Yaskawa INFORM job: ARGAZ7.JBI

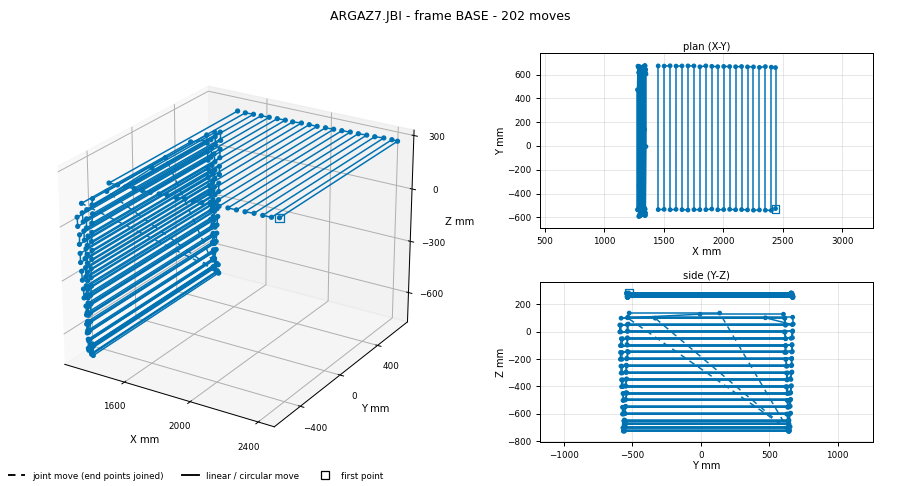
[picture p0: tool path of ARGAZ7.JBI in frame BASE, 202 of 208 moves have a stored position in this frame; points joined in program order, loops and branches not executed]
/JOB
//NAME ARGAZ7
//POS
///NPOS 202,0,202,0,0,0
///TOOL 0
///POSTYPE BASE
///RECTAN
///RCONF 1,0,0,0,0,0,0,0,0,0,0,0,0,0,0,0,0,0,0,0,0,0,0,0
C00000=2438.206271,-525.697965,282.313487,175.000000,5.000000,5.000000
C00001=2438.206271,658.166328,282.313487,175.000000,5.000000,5.000000
C00002=2403.104531,661.654143,282.437479,175.000000,5.000000,5.000000
C00003=2403.104531,-541.268813,282.437479,175.000000,5.000000,5.000000
C00004=2353.104531,-539.692706,280.280820,175.000000,5.000000,5.000000
C00005=2353.104531,666.367518,280.280820,175.000000,5.000000,5.000000
C00006=2303.104531,659.842979,278.975224,175.000000,5.000000,5.000000
C00007=2303.104531,-537.369308,278.975224,175.000000,5.000000,5.000000
C00008=2253.104531,-539.325854,276.432507,175.000000,5.000000,5.000000
C00009=2253.104531,663.877677,276.432507,175.000000,5.000000,5.000000
C00010=2203.104531,664.095750,273.988823,175.000000,5.000000,5.000000
C00011=2203.104531,-536.808159,273.988823,175.000000,5.000000,5.000000
C00012=2153.104531,-534.305410,272.087713,175.000000,5.000000,5.000000
C00013=2153.104531,667.128397,272.087713,175.000000,5.000000,5.000000
C00014=2103.104531,665.272395,270.104448,175.000000,5.000000,5.000000
C00015=2103.104531,-535.482055,270.104448,175.000000,5.000000,5.000000
C00016=2053.104531,-532.207558,267.676633,175.000000,5.000000,5.000000
C00017=2053.104531,666.894698,267.676633,175.000000,5.000000,5.000000
C00018=2003.104531,667.621610,265.646124,175.000000,5.000000,5.000000
C00019=2003.104531,-533.994265,265.646124,175.000000,5.000000,5.000000
C00020=1953.104531,-535.817658,264.262638,175.000000,5.000000,5.000000
C00021=1953.104531,665.764249,264.262638,175.000000,5.000000,5.000000
C00022=1903.104531,668.606677,262.597691,175.000000,5.000000,5.000000
C00023=1903.104531,-529.609020,262.597691,175.000000,5.000000,5.000000
C00024=1853.104531,-535.014658,260.699220,175.000000,5.000000,5.000000
C00025=1853.104531,672.443681,260.699220,175.000000,5.000000,5.000000
C00026=1803.104531,665.010164,259.433234,175.000000,5.000000,5.000000
C00027=1803.104531,-534.903244,259.433234,175.000000,5.000000,5.000000
C00028=1753.104531,-534.503782,257.000030,175.000000,5.000000,5.000000
C00029=1753.104531,672.230363,257.000030,175.000000,5.000000,5.000000
C00030=1703.104531,672.470856,255.326633,175.000000,5.000000,5.000000
C00031=1703.104531,-538.010620,255.326633,175.000000,5.000000,5.000000
C00032=1653.104531,-534.934494,253.475396,175.000000,5.000000,5.000000
C00033=1653.104531,671.829543,253.475396,175.000000,5.000000,5.000000
C00034=1603.104531,670.609419,252.672149,175.000000,5.000000,5.000000
C00035=1603.104531,-532.412044,252.672149,175.000000,5.000000,5.000000
C00036=1553.104531,-535.348902,250.461758,175.000000,5.000000,5.000000
C00037=1553.104531,673.341791,250.461758,175.000000,5.000000,5.000000
C00038=1503.104531,670.724910,249.387708,175.000000,5.000000,5.000000
C00039=1503.104531,-532.359734,249.387708,175.000000,5.000000,5.000000
C00040=1453.054088,-534.367911,249.591599,175.000000,5.000000,5.000000
C00041=1453.054088,672.087699,249.591599,175.000000,5.000000,5.000000
C00042=1350.381240,603.865126,127.297248,175.000000,-89.999999,5.000000
C00043=1350.381240,-4.872901,127.297248,175.000000,-89.999999,5.000000
C00044=1345.317967,-581.433967,98.136038,175.000000,-89.999999,5.000000
C00045=1345.317967,614.304117,98.136038,175.000000,-89.999999,5.000000
C00046=1343.165957,618.982165,48.136038,175.000000,-89.999999,5.000000
C00047=1343.165957,-582.765505,48.136038,175.000000,-89.999999,5.000000
C00048=1341.300612,-583.336165,-1.863962,175.000000,-89.999999,5.000000
C00049=1341.300612,609.146443,-1.863962,175.000000,-89.999999,5.000000
C00050=1339.709084,619.520215,-51.863962,175.000000,-89.999999,5.000000
C00051=1339.709084,-570.470513,-51.863962,175.000000,-89.999999,5.000000
C00052=1337.699081,-576.338794,-101.863962,175.000000,-89.999999,5.000000
C00053=1337.699081,621.164257,-101.863962,175.000000,-89.999999,5.000000
C00054=1336.029732,622.134378,-151.863962,175.000000,-89.999999,5.000000
C00055=1336.029732,-575.046658,-151.863962,175.000000,-89.999999,5.000000
C00056=1334.409462,-575.048017,-201.863962,175.000000,-89.999999,5.000000
C00057=1334.409462,620.847677,-201.863962,175.000000,-89.999999,5.000000
C00058=1332.613520,629.372241,-251.863962,175.000000,-89.999999,5.000000
C00059=1332.613520,-574.966494,-251.863962,175.000000,-89.999999,5.000000
C00060=1330.809111,-573.285766,-301.863962,175.000000,-89.999999,5.000000
C00061=1330.809111,633.836971,-301.863962,175.000000,-89.999999,5.000000
C00062=1328.972483,628.403479,-351.863962,175.000000,-89.999999,5.000000
C00063=1328.972483,-568.874026,-351.863962,175.000000,-89.999999,5.000000
C00064=1327.018956,-568.863156,-401.863962,175.000000,-89.999999,5.000000
C00065=1327.018956,630.494538,-401.863962,175.000000,-89.999999,5.000000
C00066=1325.088817,639.463401,-451.863962,175.000000,-89.999999,5.000000
C00067=1325.088817,-566.032958,-451.863962,175.000000,-89.999999,5.000000
C00068=1323.161118,-565.087294,-501.863962,175.000000,-89.999999,5.000000
C00069=1323.161118,635.588352,-501.863962,175.000000,-89.999999,5.000000
C00070=1321.094332,638.798990,-551.863962,175.000000,-89.999999,5.000000
C00071=1321.094332,-562.729927,-551.863962,175.000000,-89.999999,5.000000
C00072=1319.309806,-563.197324,-601.863962,175.000000,-89.999999,5.000000
C00073=1319.309806,636.908341,-601.863962,175.000000,-89.999999,5.000000
C00074=1317.380318,638.679424,-651.863962,175.000000,-89.999999,5.000000
C00075=1317.380318,-558.654468,-651.863962,175.000000,-89.999999,5.000000
C00076=1315.669137,-556.653763,-701.863962,175.000000,-89.999999,5.000000
C00077=1315.669137,640.156344,-701.863962,175.000000,-89.999999,5.000000
C00078=1334.065119,643.160458,-676.863962,180.000000,-60.000000,0.000000
C00079=1334.065119,-555.617066,-676.863962,180.000000,-60.000000,0.000000
C00080=1332.634857,-557.949975,-726.863962,180.000000,-60.000000,0.000000
C00081=1332.634857,645.315377,-726.863962,180.000000,-60.000000,0.000000
C00082=1332.634857,645.315377,-726.863962,180.000000,-60.000000,0.000000
C00083=1339.573268,138.476508,135.649167,175.000000,-89.999999,5.000000
C00084=1339.573268,-522.212780,135.649167,175.000000,-89.999999,5.000000
C00085=1342.134154,-531.684245,105.452509,175.000000,-89.999999,5.000000
C00086=1342.134154,671.005872,105.452509,175.000000,-89.999999,5.000000
C00087=1341.644946,675.400567,55.452509,175.000000,-89.999999,5.000000
C00088=1341.644946,-528.175842,55.452509,175.000000,-89.999999,5.000000
C00089=1340.416342,-534.347202,5.452509,175.000000,-89.999999,5.000000
C00090=1340.416342,670.993620,5.452509,175.000000,-89.999999,5.000000
C00091=1339.530292,669.673033,-44.547491,175.000000,-89.999999,5.000000
C00092=1339.530292,-535.215794,-44.547491,175.000000,-89.999999,5.000000
C00093=1338.211943,-538.702415,-94.547491,175.000000,-89.999999,5.000000
C00094=1338.211943,666.424662,-94.547491,175.000000,-89.999999,5.000000
C00095=1337.029328,668.773128,-144.547491,175.000000,-89.999999,5.000000
C00096=1337.029328,-535.105518,-144.547491,175.000000,-89.999999,5.000000
C00097=1335.742282,-538.419237,-194.547491,175.000000,-89.999999,5.000000
C00098=1335.742282,664.151075,-194.547491,175.000000,-89.999999,5.000000
C00099=1334.317615,664.923005,-244.547491,175.000000,-89.999999,5.000000
C00100=1334.317615,-543.588585,-244.547491,175.000000,-89.999999,5.000000
C00101=1332.622991,-545.482334,-294.547491,175.000000,-89.999999,5.000000
C00102=1332.622991,665.844693,-294.547491,175.000000,-89.999999,5.000000
C00103=1330.725701,651.986702,-344.547491,175.000000,-89.999999,5.000000
C00104=1330.725701,-540.830329,-344.547491,175.000000,-89.999999,5.000000
C00105=1328.930857,-548.962147,-394.547491,175.000000,-89.999999,5.000000
C00106=1328.930857,662.201508,-394.547491,175.000000,-89.999999,5.000000
C00107=1326.931876,657.022630,-444.547491,175.000000,-89.999999,5.000000
C00108=1326.931876,-544.291083,-444.547491,175.000000,-89.999999,5.000000
C00109=1325.288169,-548.069050,-494.547491,175.000000,-89.999999,5.000000
C00110=1325.288169,656.905547,-494.547491,175.000000,-89.999999,5.000000
C00111=1323.374017,653.466576,-544.547491,175.000000,-89.999999,5.000000
C00112=1323.374017,-547.809017,-544.547491,175.000000,-89.999999,5.000000
C00113=1321.288396,-554.990557,-594.547491,175.000000,-89.999999,5.000000
C00114=1321.288396,656.080521,-594.547491,175.000000,-89.999999,5.000000
C00115=1319.367287,642.085025,-644.547491,175.000000,-89.999999,5.000000
C00116=1319.367287,-557.326770,-644.547491,175.000000,-89.999999,5.000000
C00117=1317.423937,-557.694356,-694.547491,175.000000,-89.999999,5.000000
C00118=1317.423937,652.683754,-694.547491,175.000000,-89.999999,5.000000
C00119=1335.544484,639.032700,-669.547491,180.000000,-60.000000,0.000000
C00120=1335.544484,-553.686308,-669.547491,180.000000,-60.000000,0.000000
C00121=1333.832838,-562.636346,-719.547491,180.000000,-60.000000,0.000000
C00122=1333.832838,646.517840,-719.547491,180.000000,-60.000000,0.000000
C00123=1333.832838,646.517840,-719.547491,180.000000,-60.000000,0.000000
C00124=1279.346652,-534.805452,101.042948,175.000000,-89.999999,5.000000
C00125=1279.346652,472.104166,101.042948,175.000000,-89.999999,5.000000
C00126=1283.463175,668.476204,51.042948,175.000000,-89.999999,5.000000
C00127=1283.463175,-536.860505,51.042948,175.000000,-89.999999,5.000000
C00128=1286.233170,-534.734799,1.042948,175.000000,-89.999999,5.000000
C00129=1286.233170,670.246607,1.042948,175.000000,-89.999999,5.000000
C00130=1288.530819,659.150000,-48.957052,175.000000,-89.999999,5.000000
C00131=1288.530819,-534.611156,-48.957052,175.000000,-89.999999,5.000000
C00132=1290.803481,-535.551386,-98.957052,175.000000,-89.999999,5.000000
C00133=1290.803481,666.067207,-98.957052,175.000000,-89.999999,5.000000
C00134=1293.209386,664.711211,-148.957052,175.000000,-89.999999,5.000000
C00135=1293.209386,-527.270031,-148.957052,175.000000,-89.999999,5.000000
C00136=1294.839574,-540.608514,-198.957052,175.000000,-89.999999,5.000000
C00137=1294.839574,663.751960,-198.957052,175.000000,-89.999999,5.000000
C00138=1296.633537,661.020947,-248.957052,175.000000,-89.999999,5.000000
C00139=1296.633537,-540.046007,-248.957052,175.000000,-89.999999,5.000000
C00140=1298.209048,-543.528388,-298.957052,175.000000,-89.999999,5.000000
C00141=1298.209048,662.091613,-298.957052,175.000000,-89.999999,5.000000
C00142=1299.776483,658.821192,-348.957052,175.000000,-89.999999,5.000000
C00143=1299.776483,-543.652031,-348.957052,175.000000,-89.999999,5.000000
C00144=1301.502905,-546.906148,-398.957052,175.000000,-89.999999,5.000000
C00145=1301.502905,658.989672,-398.957052,175.000000,-89.999999,5.000000
C00146=1302.998852,654.262710,-448.957052,175.000000,-89.999999,5.000000
C00147=1302.998852,-537.101677,-448.957052,175.000000,-89.999999,5.000000
C00148=1304.424846,-550.182005,-498.957052,175.000000,-89.999999,5.000000
C00149=1304.424846,652.394480,-498.957052,175.000000,-89.999999,5.000000
C00150=1305.126958,645.352272,-548.957052,175.000000,-89.999999,5.000000
C00151=1305.126958,-549.584171,-548.957052,175.000000,-89.999999,5.000000
C00152=1306.384029,-551.767622,-598.957052,175.000000,-89.999999,5.000000
C00153=1306.384029,652.495025,-598.957052,175.000000,-89.999999,5.000000
C00154=1307.818366,644.325085,-648.957052,175.000000,-89.999999,5.000000
C00155=1307.818366,-551.682023,-648.957052,175.000000,-89.999999,5.000000
C00156=1309.126713,-554.874998,-698.957052,175.000000,-89.999999,5.000000
C00157=1309.126713,646.027552,-698.957052,175.000000,-89.999999,5.000000
C00158=1330.557262,644.373999,-673.957052,180.000000,-60.000000,0.000000
C00159=1330.557262,-546.749896,-673.957052,180.000000,-60.000000,0.000000
C00160=1331.629790,-555.586964,-723.957052,180.000000,-60.000000,0.000000
C00161=1331.629790,642.223156,-723.957052,180.000000,-60.000000,0.000000
C00162=1331.629790,642.223156,-723.957052,180.000000,-60.000000,0.000000
C00163=1292.184949,-332.258153,98.133784,175.000000,-89.999999,5.000000
C00164=1292.184949,612.097991,98.133784,175.000000,-89.999999,5.000000
C00165=1290.843307,617.746562,48.133784,175.000000,-89.999999,5.000000
C00166=1290.843307,-591.020978,48.133784,175.000000,-89.999999,5.000000
C00167=1292.718404,-590.852160,-1.866216,175.000000,-89.999999,5.000000
C00168=1292.718404,617.113497,-1.866216,175.000000,-89.999999,5.000000
C00169=1294.622390,619.663454,-51.866216,175.000000,-89.999999,5.000000
C00170=1294.622390,-579.746980,-51.866216,175.000000,-89.999999,5.000000
C00171=1296.401213,-586.430237,-101.866216,175.000000,-89.999999,5.000000
C00172=1296.401213,618.745851,-101.866216,175.000000,-89.999999,5.000000
C00173=1298.367894,613.365481,-151.866216,175.000000,-89.999999,5.000000
C00174=1298.367894,-585.535778,-151.866216,175.000000,-89.999999,5.000000
C00175=1300.139338,-586.488779,-201.866216,175.000000,-89.999999,5.000000
C00176=1300.139338,622.021450,-201.866216,175.000000,-89.999999,5.000000
C00177=1301.999434,624.889982,-251.866216,175.000000,-89.999999,5.000000
C00178=1301.999434,-582.499790,-251.866216,175.000000,-89.999999,5.000000
C00179=1304.062129,-581.254082,-301.866216,175.000000,-89.999999,5.000000
C00180=1304.062129,625.841622,-301.866216,175.000000,-89.999999,5.000000
C00181=1306.582167,630.514048,-351.866216,175.000000,-89.999999,5.000000
C00182=1306.582167,-577.829406,-351.866216,175.000000,-89.999999,5.000000
C00183=1308.639708,-577.839617,-401.866216,175.000000,-89.999999,5.000000
C00184=1308.639708,621.578986,-401.866216,175.000000,-89.999999,5.000000
C00185=1310.975004,631.745461,-451.866216,175.000000,-89.999999,5.000000
C00186=1310.975004,-566.829736,-451.866216,175.000000,-89.999999,5.000000
C00187=1313.177801,-566.867856,-501.866216,175.000000,-89.999999,5.000000
C00188=1313.177801,631.511295,-501.866216,175.000000,-89.999999,5.000000
C00189=1315.115577,634.444495,-551.866216,175.000000,-89.999999,5.000000
C00190=1315.115577,-571.282972,-551.866216,175.000000,-89.999999,5.000000
C00191=1317.145755,-571.372827,-601.866216,175.000000,-89.999999,5.000000
C00192=1317.145755,627.765321,-601.866216,175.000000,-89.999999,5.000000
C00193=1319.380465,638.267389,-651.866216,175.000000,-89.999999,5.000000
C00194=1319.380465,-561.885024,-651.866216,175.000000,-89.999999,5.000000
C00195=1321.674662,-568.241539,-701.866216,175.000000,-89.999999,5.000000
C00196=1321.674662,630.219979,-701.866216,175.000000,-89.999999,5.000000
C00197=1343.978496,641.568175,-676.866216,180.000000,-60.000000,0.000000
C00198=1343.978496,-559.132214,-676.866216,180.000000,-60.000000,0.000000
C00199=1346.283422,-564.960494,-726.866216,180.000000,-60.000000,0.000000
C00200=1346.283422,641.391869,-726.866216,180.000000,-60.000000,0.000000
C00201=1346.283422,641.391869,-726.866216,180.000000,-60.000000,0.000000
///POSTYPE PULSE
///PULSE
EC00000=0
EC00001=0
EC00002=0
EC00003=0
EC00004=0
EC00005=0
EC00006=0
EC00007=0
EC00008=0
EC00009=0
EC00010=0
EC00011=0
EC00012=0
EC00013=0
EC00014=0
EC00015=0
EC00016=0
EC00017=0
EC00018=0
EC00019=0
EC00020=0
EC00021=0
EC00022=0
EC00023=0
EC00024=0
EC00025=0
EC00026=0
EC00027=0
EC00028=0
EC00029=0
EC00030=0
EC00031=0
EC00032=0
EC00033=0
EC00034=0
EC00035=0
EC00036=0
EC00037=0
EC00038=0
EC00039=0
EC00040=0
EC00041=0
EC00042=0
EC00043=0
EC00044=0
EC00045=0
EC00046=0
EC00047=0
EC00048=0
EC00049=0
EC00050=0
EC00051=0
EC00052=0
EC00053=0
EC00054=0
EC00055=0
EC00056=0
EC00057=0
EC00058=0
EC00059=0
EC00060=0
EC00061=0
EC00062=0
EC00063=0
EC00064=0
EC00065=0
EC00066=0
EC00067=0
EC00068=0
EC00069=0
EC00070=0
EC00071=0
EC00072=0
EC00073=0
EC00074=0
EC00075=0
EC00076=0
EC00077=0
EC00078=0
EC00079=0
EC00080=0
EC00081=0
EC00082=92160
EC00083=92160
EC00084=92160
EC00085=92160
EC00086=92160
EC00087=92160
EC00088=92160
EC00089=92160
EC00090=92160
EC00091=92160
EC00092=92160
EC00093=92160
EC00094=92160
EC00095=92160
EC00096=92160
EC00097=92160
EC00098=92160
EC00099=92160
EC00100=92160
EC00101=92160
EC00102=92160
EC00103=92160
EC00104=92160
EC00105=92160
EC00106=92160
EC00107=92160
EC00108=92160
EC00109=92160
EC00110=92160
EC00111=92160
EC00112=92160
EC00113=92160
EC00114=92160
EC00115=92160
EC00116=92160
EC00117=92160
EC00118=92160
EC00119=92160
EC00120=92160
EC00121=92160
EC00122=92160
EC00123=184320
EC00124=184320
EC00125=184320
EC00126=184320
EC00127=184320
EC00128=184320
EC00129=184320
EC00130=184320
EC00131=184320
EC00132=184320
EC00133=184320
EC00134=184320
EC00135=184320
EC00136=184320
EC00137=184320
EC00138=184320
EC00139=184320
EC00140=184320
EC00141=184320
EC00142=184320
EC00143=184320
EC00144=184320
EC00145=184320
EC00146=184320
EC00147=184320
EC00148=184320
EC00149=184320
EC00150=184320
EC00151=184320
EC00152=184320
EC00153=184320
EC00154=184320
EC00155=184320
EC00156=184320
EC00157=184320
EC00158=184320
EC00159=184320
EC00160=184320
EC00161=184320
EC00162=276480
EC00163=276480
EC00164=276480
EC00165=276480
EC00166=276480
EC00167=276480
EC00168=276480
EC00169=276480
EC00170=276480
EC00171=276480
EC00172=276480
EC00173=276480
EC00174=276480
EC00175=276480
EC00176=276480
EC00177=276480
EC00178=276480
EC00179=276480
EC00180=276480
EC00181=276480
EC00182=276480
EC00183=276480
EC00184=276480
EC00185=276480
EC00186=276480
EC00187=276480
EC00188=276480
EC00189=276480
EC00190=276480
EC00191=276480
EC00192=276480
EC00193=276480
EC00194=276480
EC00195=276480
EC00196=276480
EC00197=276480
EC00198=276480
EC00199=276480
EC00200=276480
EC00201=368640
//INST
///DATE 2023/01/30 13:49
///ATTR SC,RW,RJ
////FRAME BASE
///GROUP1 RB1,ST1
NOP
MOVJ P009 EX000 VJ=15.00
MOVJ C00000 EC00000 VJ=12.0
CALL JOB:SPYON
MOVL C00001 EC00001 V=150.0
MOVL C00002 EC00002 V=150.0
MOVL C00003 EC00003 V=150.0
MOVL C00004 EC00004 V=150.0
MOVL C00005 EC00005 V=150.0
MOVL C00006 EC00006 V=150.0
MOVL C00007 EC00007 V=150.0
MOVL C00008 EC00008 V=150.0
MOVL C00009 EC00009 V=150.0
MOVL C00010 EC00010 V=150.0
MOVL C00011 EC00011 V=150.0
MOVL C00012 EC00012 V=150.0
MOVL C00013 EC00013 V=150.0
MOVL C00014 EC00014 V=150.0
MOVL C00015 EC00015 V=150.0
MOVL C00016 EC00016 V=150.0
MOVL C00017 EC00017 V=150.0
MOVL C00018 EC00018 V=150.0
MOVL C00019 EC00019 V=150.0
MOVL C00020 EC00020 V=150.0
MOVL C00021 EC00021 V=150.0
MOVL C00022 EC00022 V=150.0
MOVL C00023 EC00023 V=150.0
MOVL C00024 EC00024 V=150.0
MOVL C00025 EC00025 V=150.0
MOVL C00026 EC00026 V=150.0
MOVL C00027 EC00027 V=150.0
MOVL C00028 EC00028 V=150.0
MOVL C00029 EC00029 V=150.0
MOVL C00030 EC00030 V=150.0
MOVL C00031 EC00031 V=150.0
MOVL C00032 EC00032 V=150.0
MOVL C00033 EC00033 V=150.0
MOVL C00034 EC00034 V=150.0
MOVL C00035 EC00035 V=150.0
MOVL C00036 EC00036 V=150.0
MOVL C00037 EC00037 V=150.0
MOVL C00038 EC00038 V=150.0
MOVL C00039 EC00039 V=150.0
MOVL C00040 EC00040 V=150.0
MOVL C00041 EC00041 V=150.0
CALL JOB:SPYOF
MOVJ P009 VJ=15.00
MOVJ C00042 EC00042 VJ=12.0
CALL JOB:SPYON
MOVL C00043 EC00043 V=150.0
MOVL C00044 EC00044 V=150.0
MOVL C00045 EC00045 V=150.0
MOVL C00046 EC00046 V=150.0
MOVL C00047 EC00047 V=150.0
MOVL C00048 EC00048 V=150.0
MOVL C00049 EC00049 V=150.0
MOVL C00050 EC00050 V=150.0
MOVL C00051 EC00051 V=150.0
MOVL C00052 EC00052 V=150.0
MOVL C00053 EC00053 V=150.0
MOVL C00054 EC00054 V=150.0
MOVL C00055 EC00055 V=150.0
MOVL C00056 EC00056 V=150.0
MOVL C00057 EC00057 V=150.0
MOVL C00058 EC00058 V=150.0
MOVL C00059 EC00059 V=150.0
MOVL C00060 EC00060 V=150.0
MOVL C00061 EC00061 V=150.0
MOVL C00062 EC00062 V=150.0
MOVL C00063 EC00063 V=150.0
MOVL C00064 EC00064 V=150.0
MOVL C00065 EC00065 V=150.0
MOVL C00066 EC00066 V=150.0
MOVL C00067 EC00067 V=150.0
MOVL C00068 EC00068 V=150.0
MOVL C00069 EC00069 V=150.0
MOVL C00070 EC00070 V=150.0
MOVL C00071 EC00071 V=150.0
MOVL C00072 EC00072 V=150.0
MOVL C00073 EC00073 V=150.0
MOVL C00074 EC00074 V=150.0
MOVL C00075 EC00075 V=150.0
MOVL C00076 EC00076 V=150.0
MOVL C00077 EC00077 V=150.0
MOVL C00078 EC00078 V=150.0
MOVL C00079 EC00079 V=150.0
MOVL C00080 EC00080 V=150.0
MOVL C00081 EC00081 V=150.0
CALL JOB:SPYOF
MOVJ P009 VJ=15.00
MOVL C00082 EC00082 V=150.0
MOVJ C00083 EC00083 VJ=12.0
CALL JOB:SPYON
MOVL C00084 EC00084 V=150.0
MOVL C00085 EC00085 V=150.0
MOVL C00086 EC00086 V=150.0
MOVL C00087 EC00087 V=150.0
MOVL C00088 EC00088 V=150.0
MOVL C00089 EC00089 V=150.0
MOVL C00090 EC00090 V=150.0
MOVL C00091 EC00091 V=150.0
MOVL C00092 EC00092 V=150.0
MOVL C00093 EC00093 V=150.0
MOVL C00094 EC00094 V=150.0
MOVL C00095 EC00095 V=150.0
MOVL C00096 EC00096 V=150.0
MOVL C00097 EC00097 V=150.0
MOVL C00098 EC00098 V=150.0
MOVL C00099 EC00099 V=150.0
MOVL C00100 EC00100 V=150.0
MOVL C00101 EC00101 V=150.0
MOVL C00102 EC00102 V=150.0
MOVL C00103 EC00103 V=150.0
MOVL C00104 EC00104 V=150.0
MOVL C00105 EC00105 V=150.0
MOVL C00106 EC00106 V=150.0
MOVL C00107 EC00107 V=150.0
MOVL C00108 EC00108 V=150.0
MOVL C00109 EC00109 V=150.0
MOVL C00110 EC00110 V=150.0
MOVL C00111 EC00111 V=150.0
MOVL C00112 EC00112 V=150.0
MOVL C00113 EC00113 V=150.0
MOVL C00114 EC00114 V=150.0
MOVL C00115 EC00115 V=150.0
MOVL C00116 EC00116 V=150.0
MOVL C00117 EC00117 V=150.0
MOVL C00118 EC00118 V=150.0
MOVL C00119 EC00119 V=150.0
MOVL C00120 EC00120 V=150.0
MOVL C00121 EC00121 V=150.0
MOVL C00122 EC00122 V=150.0
CALL JOB:SPYOF
MOVJ P009 VJ=15.00
MOVL C00123 EC00123 V=150.0
MOVJ C00124 EC00124 VJ=12.0
CALL JOB:SPYON
MOVL C00125 EC00125 V=150.0
MOVL C00126 EC00126 V=150.0
MOVL C00127 EC00127 V=150.0
MOVL C00128 EC00128 V=150.0
MOVL C00129 EC00129 V=150.0
MOVL C00130 EC00130 V=150.0
MOVL C00131 EC00131 V=150.0
MOVL C00132 EC00132 V=150.0
MOVL C00133 EC00133 V=150.0
MOVL C00134 EC00134 V=150.0
MOVL C00135 EC00135 V=150.0
MOVL C00136 EC00136 V=150.0
MOVL C00137 EC00137 V=150.0
MOVL C00138 EC00138 V=150.0
MOVL C00139 EC00139 V=150.0
MOVL C00140 EC00140 V=150.0
MOVL C00141 EC00141 V=150.0
MOVL C00142 EC00142 V=150.0
MOVL C00143 EC00143 V=150.0
MOVL C00144 EC00144 V=150.0
MOVL C00145 EC00145 V=150.0
MOVL C00146 EC00146 V=150.0
MOVL C00147 EC00147 V=150.0
MOVL C00148 EC00148 V=150.0
MOVL C00149 EC00149 V=150.0
MOVL C00150 EC00150 V=150.0
MOVL C00151 EC00151 V=150.0
MOVL C00152 EC00152 V=150.0
MOVL C00153 EC00153 V=150.0
MOVL C00154 EC00154 V=150.0
MOVL C00155 EC00155 V=150.0
MOVL C00156 EC00156 V=150.0
MOVL C00157 EC00157 V=150.0
MOVL C00158 EC00158 V=150.0
MOVL C00159 EC00159 V=150.0
MOVL C00160 EC00160 V=150.0
MOVL C00161 EC00161 V=150.0
CALL JOB:SPYOF
MOVJ P009 VJ=15.00
MOVL C00162 EC00162 V=150.0
MOVJ C00163 EC00163 VJ=12.0
CALL JOB:SPYON
MOVL C00164 EC00164 V=150.0
MOVL C00165 EC00165 V=150.0
MOVL C00166 EC00166 V=150.0
MOVL C00167 EC00167 V=150.0
MOVL C00168 EC00168 V=150.0
MOVL C00169 EC00169 V=150.0
MOVL C00170 EC00170 V=150.0
MOVL C00171 EC00171 V=150.0
MOVL C00172 EC00172 V=150.0
MOVL C00173 EC00173 V=150.0
MOVL C00174 EC00174 V=150.0
MOVL C00175 EC00175 V=150.0
MOVL C00176 EC00176 V=150.0
MOVL C00177 EC00177 V=150.0
MOVL C00178 EC00178 V=150.0
MOVL C00179 EC00179 V=150.0
MOVL C00180 EC00180 V=150.0
MOVL C00181 EC00181 V=150.0
MOVL C00182 EC00182 V=150.0
MOVL C00183 EC00183 V=150.0
MOVL C00184 EC00184 V=150.0
MOVL C00185 EC00185 V=150.0
MOVL C00186 EC00186 V=150.0
MOVL C00187 EC00187 V=150.0
MOVL C00188 EC00188 V=150.0
MOVL C00189 EC00189 V=150.0
MOVL C00190 EC00190 V=150.0
MOVL C00191 EC00191 V=150.0
MOVL C00192 EC00192 V=150.0
MOVL C00193 EC00193 V=150.0
MOVL C00194 EC00194 V=150.0
MOVL C00195 EC00195 V=150.0
MOVL C00196 EC00196 V=150.0
MOVL C00197 EC00197 V=150.0
MOVL C00198 EC00198 V=150.0
MOVL C00199 EC00199 V=150.0
MOVL C00200 EC00200 V=150.0
CALL JOB:SPYOF
MOVJ P009 VJ=15.00
MOVL C00201 EC00201 V=150.0
END
